PROGRAM POU
VAR
END_VAR

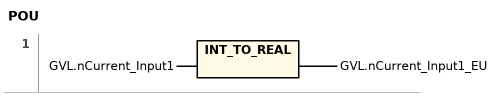
// NETWORK 1
GVL.nCurrent_Input1_EU := INT_TO_REAL(GVL.nCurrent_Input1);

END_PROGRAM

(* stored: Version 1.1.0.1, ProductVersion 3.1.4024.12
   POU POU: Id {a5aab107-3d17-4a4d-af9d-3cc7e73d8153}, SpecialFunc None *)
